{attribute 'no_explicit_call':= 'do not call this POU directly'}
FUNCTION_BLOCK T_StructureMonitor
VAR
    _Changed   : BOOL;
    Stored_CRC : WORD := 16#FFFF;
END_VAR

PROPERTY Changed : BOOL
GET
Changed := _Changed;
END_GET
END_PROPERTY

METHOD Reset
VAR_INPUT
END_VAR
Stored_CRC := 16#FFFF;
END_METHOD

METHOD Test
VAR_INPUT
    StructureAddress : POINTER TO BYTE;
    StructureSize    : UDINT;
END_VAR
VAR
    CRC : WORD;
END_VAR
CRC := F_DATA_TO_CRC16_CCITT(pData  := StructureAddress,
                             cbData := StructureSize,
                             crc    := 0);

_Changed := (CRC <> Stored_CRC);

IF Changed THEN
    Stored_CRC := CRC;
END_IF
END_METHOD

END_FUNCTION_BLOCK

(* stored: Version 1.1.0.1, ProductVersion 3.1.4024.12
   POU T_StructureMonitor: Id {4ff37301-51db-0d33-1801-69eaef5746f6}, SpecialFunc None
   Property Changed: Id {b58d1fdb-bd27-0669-252f-03a922d82a2c}
   Get Get: Id {1abfd3ce-79a9-0f67-2fbb-cb772335c15a}
   Method Reset: Id {68db21ce-aedd-0b3b-35b4-c6242b4cf77c}
   Method Test: Id {4f5aa998-1605-0b49-0b94-abed0a451d48} *)
